TYPE ST_DriveStatus :
STRUCT
	nActLength	: UINT;
	nMaxLength	: UINT;
	strStatus	: STRING;
END_STRUCT
END_TYPE

(* stored: Version 1.1.0.1
   DUT ST_DriveStatus: Id {989ebcf2-6120-40f9-a5ee-6c9554ace2a2} *)
